(* PLC project plan_voie_railml, OpenIXl generator OpenIXL generator v0.1 *)
(* stored: companyURL https://github.com/Bleebop/IXL_project, creationDateTime 2026-09-27T16:06:12, modificationDateTime 2026-09-27T16:06:12 *)

TYPE TC : (NIL := -1, CDV10 := 1, CDV8 := 2, CDV6 := 3, CDV7 := 4, CDV9 := 5, CDV11 := 6, CDV13 := 7, CDV14 := 8, CDV12 := 9);
END_TYPE

TYPE SWITCH : (NIL := -1, SW2 := 1, SW1 := 2);
END_TYPE

TYPE SIGNAL : (NIL := -1, MRK13 := 1, MRK14 := 2, MRK15 := 3, MRK16 := 4);
END_TYPE

TYPE TRAIN_STATE : STRUCT
  exists : BOOL;
  rear_pos : TC;
  front_pos : TC;
  orientation : DIR;
  stopped : BOOL;
END_STRUCT;
END_TYPE

TYPE DIR : (NIL := -1, DOWN := 0, UP := 1);
END_TYPE

TYPE SW_POS_t : (NIL := -1, LEFT := 1, RIGHT := 2, INTERMEDIATE := 3);
END_TYPE

TYPE ENTRY_POINT_t : STRUCT
  tc : TC;
  orientation : DIR;
END_STRUCT;
END_TYPE

TYPE EXIT_POINT_t : STRUCT
  tc : TC;
  orientation : DIR;
END_STRUCT;
END_TYPE

TYPE ROUTE : (NIL := -1, ROUTE1 := 1, ROUTE2 := 2, ROUTE3 := 3);
END_TYPE

PROGRAM safety_PLC
  VAR
    route_state : ARRAY[1..const_g.nRoute] OF route_state;
    Approaching_train : ARRAY[1..const_g.nRoute] OF Approaching_train;
    switch_locked : ARRAY[1..const_g.nSwitch] OF BOOL;
    switch_required_left : ARRAY[1..const_g.nSwitch] OF BOOL;
    switch_required_right : ARRAY[1..const_g.nSwitch] OF BOOL;
  END_VAR
  VAR CONSTANT
    DELAY_DESTRUCT : ARRAY[1..const_g.nRoute] OF TIME := [TIME#99999s0ms, TIME#99999s0ms, TIME#99999s0ms];
  END_VAR
  VAR_OUTPUT
    route_open : ARRAY[1..const_g.nRoute] OF BOOL;
    route_entry_authorization : ARRAY[1..const_g.nRoute] OF BOOL;  (* The starting signal of the route can be opened to go through this route *)
    signal_open_maneuver : ARRAY[1..const_g.nSignal] OF BOOL;  (* Signal is opened for CBTC trains (downstream block occupation is ignored) *)
    switch_command_left : ARRAY[1..const_g.nSwitch] OF BOOL;
    switch_command_right : ARRAY[1..const_g.nSwitch] OF BOOL;
  END_VAR

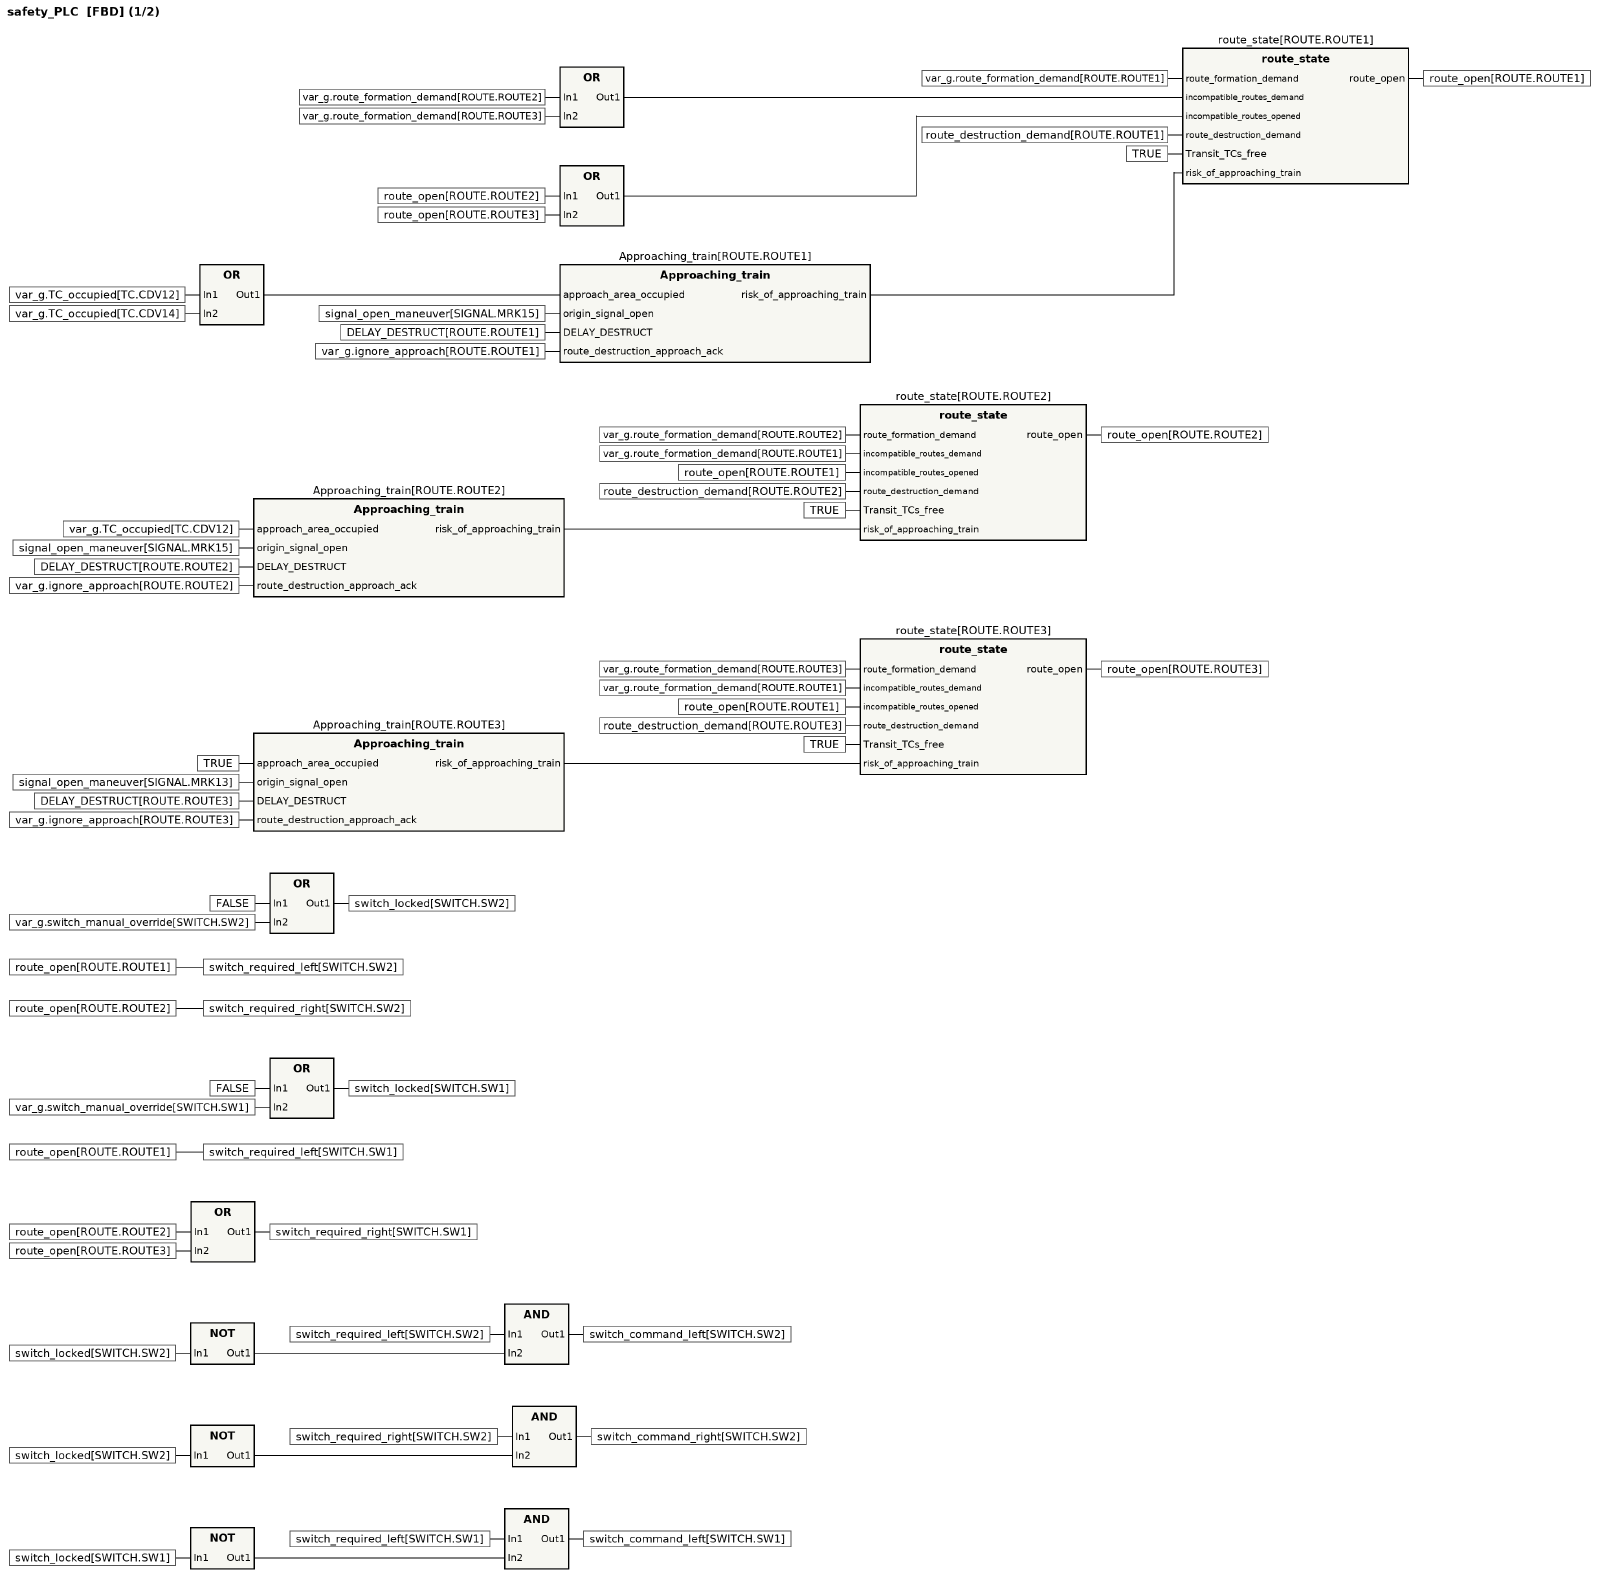
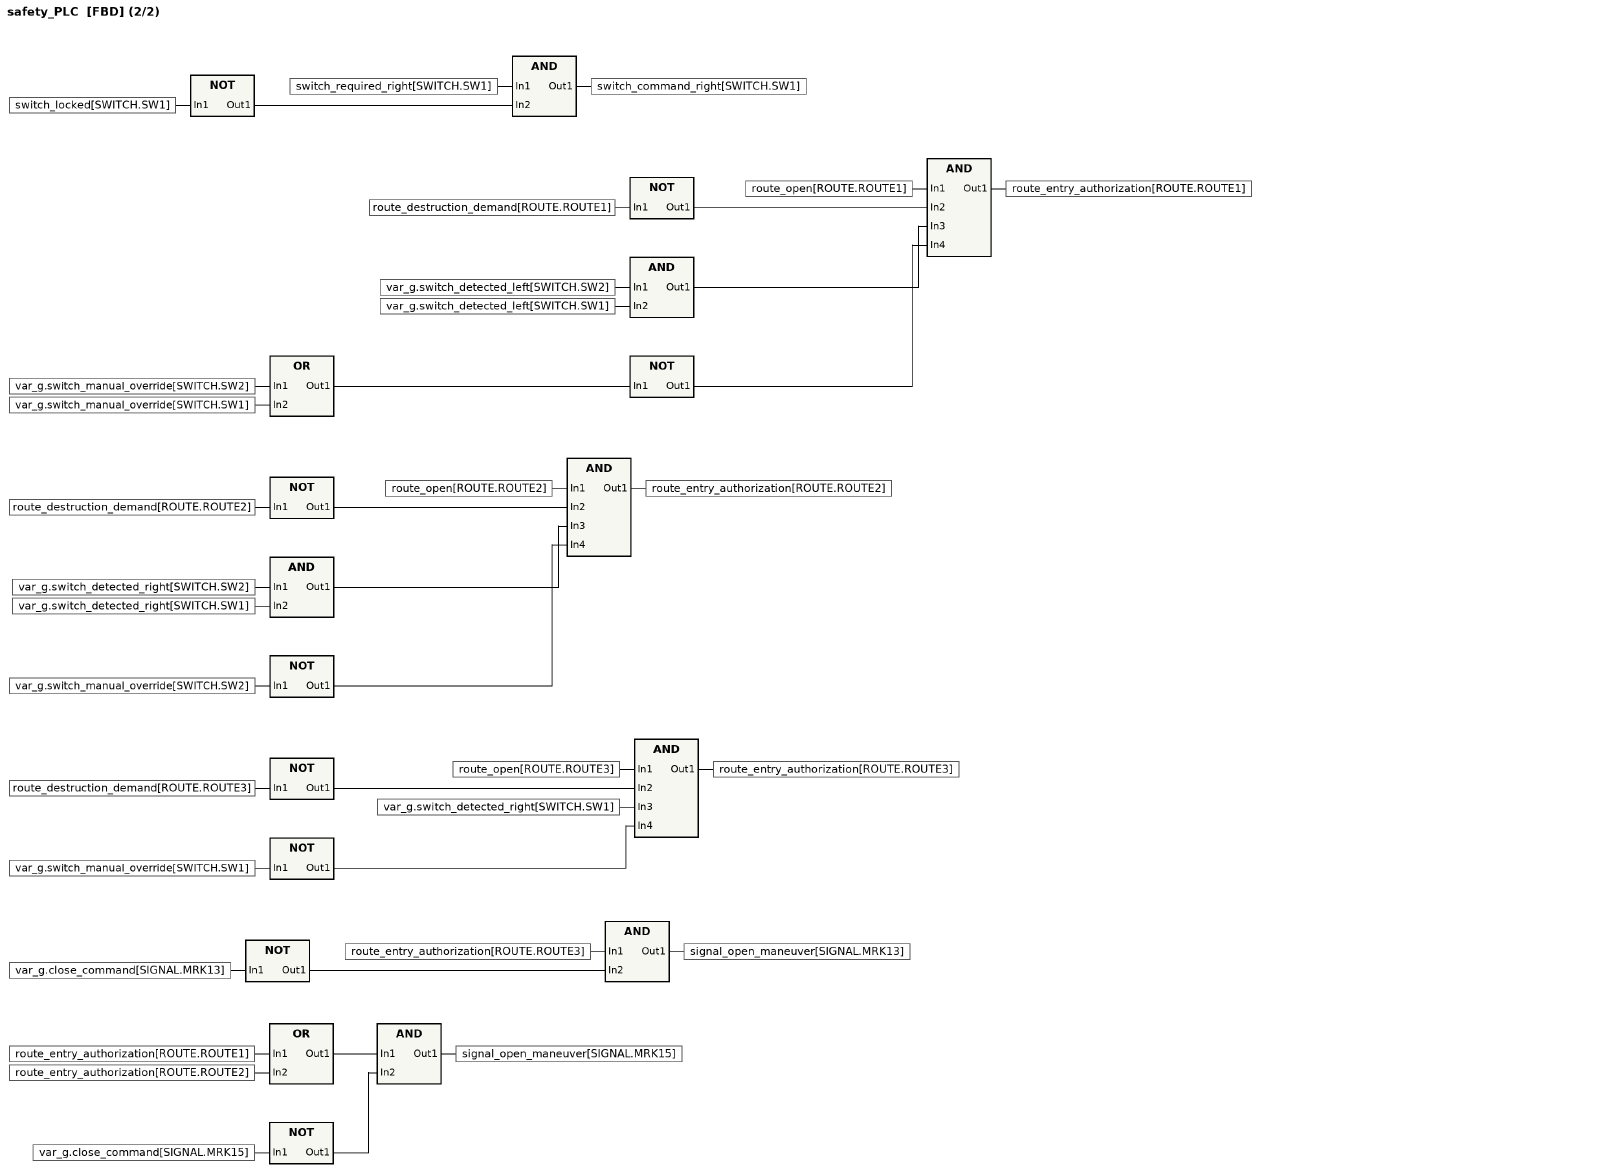
(* FBD diagram, written out as Structured Text *)
Approaching_train[ROUTE.ROUTE1](approach_area_occupied := var_g.TC_occupied[TC.CDV12] OR var_g.TC_occupied[TC.CDV14], origin_signal_open := signal_open_maneuver[SIGNAL.MRK15], DELAY_DESTRUCT := DELAY_DESTRUCT[ROUTE.ROUTE1], route_destruction_approach_ack := var_g.ignore_approach[ROUTE.ROUTE1]);
route_state[ROUTE.ROUTE1](route_formation_demand := var_g.route_formation_demand[ROUTE.ROUTE1], incompatible_routes_demand := var_g.route_formation_demand[ROUTE.ROUTE2] OR var_g.route_formation_demand[ROUTE.ROUTE3], incompatible_routes_opened := route_open[ROUTE.ROUTE2] OR route_open[ROUTE.ROUTE3], route_destruction_demand := route_destruction_demand[ROUTE.ROUTE1], Transit_TCs_free := TRUE, risk_of_approaching_train := Approaching_train[ROUTE.ROUTE1].risk_of_approaching_train);
route_open[ROUTE.ROUTE1] := route_state[ROUTE.ROUTE1].route_open;
Approaching_train[ROUTE.ROUTE2](approach_area_occupied := var_g.TC_occupied[TC.CDV12], origin_signal_open := signal_open_maneuver[SIGNAL.MRK15], DELAY_DESTRUCT := DELAY_DESTRUCT[ROUTE.ROUTE2], route_destruction_approach_ack := var_g.ignore_approach[ROUTE.ROUTE2]);
route_state[ROUTE.ROUTE2](route_formation_demand := var_g.route_formation_demand[ROUTE.ROUTE2], incompatible_routes_demand := var_g.route_formation_demand[ROUTE.ROUTE1], incompatible_routes_opened := route_open[ROUTE.ROUTE1], route_destruction_demand := route_destruction_demand[ROUTE.ROUTE2], Transit_TCs_free := TRUE, risk_of_approaching_train := Approaching_train[ROUTE.ROUTE2].risk_of_approaching_train);
route_open[ROUTE.ROUTE2] := route_state[ROUTE.ROUTE2].route_open;
Approaching_train[ROUTE.ROUTE3](approach_area_occupied := TRUE, origin_signal_open := signal_open_maneuver[SIGNAL.MRK13], DELAY_DESTRUCT := DELAY_DESTRUCT[ROUTE.ROUTE3], route_destruction_approach_ack := var_g.ignore_approach[ROUTE.ROUTE3]);
route_state[ROUTE.ROUTE3](route_formation_demand := var_g.route_formation_demand[ROUTE.ROUTE3], incompatible_routes_demand := var_g.route_formation_demand[ROUTE.ROUTE1], incompatible_routes_opened := route_open[ROUTE.ROUTE1], route_destruction_demand := route_destruction_demand[ROUTE.ROUTE3], Transit_TCs_free := TRUE, risk_of_approaching_train := Approaching_train[ROUTE.ROUTE3].risk_of_approaching_train);
route_open[ROUTE.ROUTE3] := route_state[ROUTE.ROUTE3].route_open;
switch_locked[SWITCH.SW2] := FALSE OR var_g.switch_manual_override[SWITCH.SW2];
switch_required_left[SWITCH.SW2] := route_open[ROUTE.ROUTE1];
switch_required_right[SWITCH.SW2] := route_open[ROUTE.ROUTE2];
switch_locked[SWITCH.SW1] := FALSE OR var_g.switch_manual_override[SWITCH.SW1];
switch_required_left[SWITCH.SW1] := route_open[ROUTE.ROUTE1];
switch_required_right[SWITCH.SW1] := route_open[ROUTE.ROUTE2] OR route_open[ROUTE.ROUTE3];
switch_command_left[SWITCH.SW2] := switch_required_left[SWITCH.SW2] AND NOT switch_locked[SWITCH.SW2];
switch_command_right[SWITCH.SW2] := switch_required_right[SWITCH.SW2] AND NOT switch_locked[SWITCH.SW2];
switch_command_left[SWITCH.SW1] := switch_required_left[SWITCH.SW1] AND NOT switch_locked[SWITCH.SW1];
switch_command_right[SWITCH.SW1] := switch_required_right[SWITCH.SW1] AND NOT switch_locked[SWITCH.SW1];
route_entry_authorization[ROUTE.ROUTE1] := route_open[ROUTE.ROUTE1] AND NOT route_destruction_demand[ROUTE.ROUTE1] AND var_g.switch_detected_left[SWITCH.SW2] AND var_g.switch_detected_left[SWITCH.SW1] AND NOT (var_g.switch_manual_override[SWITCH.SW2] OR var_g.switch_manual_override[SWITCH.SW1]);
route_entry_authorization[ROUTE.ROUTE2] := route_open[ROUTE.ROUTE2] AND NOT route_destruction_demand[ROUTE.ROUTE2] AND var_g.switch_detected_right[SWITCH.SW2] AND var_g.switch_detected_right[SWITCH.SW1] AND NOT var_g.switch_manual_override[SWITCH.SW2];
route_entry_authorization[ROUTE.ROUTE3] := route_open[ROUTE.ROUTE3] AND NOT route_destruction_demand[ROUTE.ROUTE3] AND var_g.switch_detected_right[SWITCH.SW1] AND NOT var_g.switch_manual_override[SWITCH.SW1];
signal_open_maneuver[SIGNAL.MRK13] := route_entry_authorization[ROUTE.ROUTE3] AND NOT var_g.close_command[SIGNAL.MRK13];
signal_open_maneuver[SIGNAL.MRK15] := (route_entry_authorization[ROUTE.ROUTE1] OR route_entry_authorization[ROUTE.ROUTE2]) AND NOT var_g.close_command[SIGNAL.MRK15];
END_PROGRAM

FUNCTION_BLOCK route_state
  VAR_INPUT
    route_formation_demand : BOOL;
    incompatible_routes_demand : BOOL;
    incompatible_routes_opened : BOOL;
    route_destruction_demand : BOOL;
    Transit_TCs_free : BOOL;
    risk_of_approaching_train : BOOL;
  END_VAR
  VAR
    SR_route : SR;
  END_VAR
  VAR_OUTPUT
    route_open : BOOL;
  END_VAR

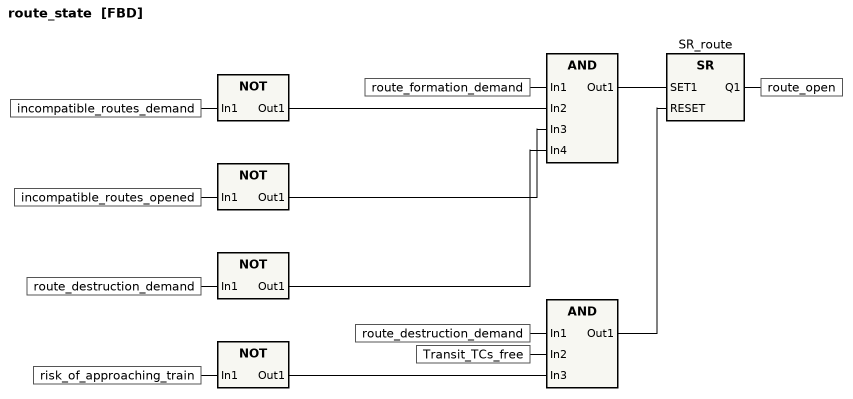
(* FBD diagram, written out as Structured Text *)
SR_route(SET1 := route_formation_demand AND NOT incompatible_routes_demand AND NOT incompatible_routes_opened AND NOT route_destruction_demand, RESET := route_destruction_demand AND Transit_TCs_free AND NOT risk_of_approaching_train);
route_open := SR_route.Q1;
END_FUNCTION_BLOCK

FUNCTION_BLOCK Approaching_train
  VAR_INPUT
    approach_area_occupied : BOOL;
    origin_signal_open : BOOL;
    DELAY_DESTRUCT : TIME;
    route_destruction_approach_ack : BOOL;
  END_VAR
  VAR_OUTPUT
    risk_of_approaching_train : BOOL;
  END_VAR
  VAR
    TON_approach_timer : TON;
    SR_approaching_train : SR;
  END_VAR

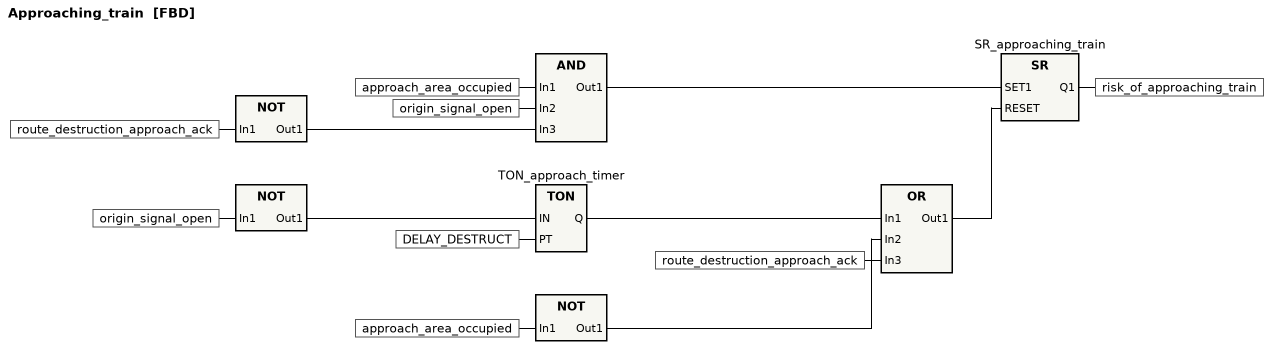
(* FBD diagram, written out as Structured Text *)
TON_approach_timer(IN := NOT origin_signal_open, PT := DELAY_DESTRUCT);
SR_approaching_train(SET1 := approach_area_occupied AND origin_signal_open AND NOT route_destruction_approach_ack, RESET := TON_approach_timer.Q OR NOT approach_area_occupied OR route_destruction_approach_ack);
risk_of_approaching_train := SR_approaching_train.Q1;
END_FUNCTION_BLOCK

CONFIGURATION Device
  RESOURCE Application ON PLC
    VAR_GLOBAL  (* var_g *)
      TC_occupied : ARRAY[1..const_g.nTC] OF BOOL;  (* /!\ safety critical /!\ *)
      switch_detected_left : ARRAY[1..const_g.nSwitch] OF BOOL;  (* /!\ safety critical /!\ *)
      switch_detected_right : ARRAY[1..const_g.nSwitch] OF BOOL;  (* /!\ safety critical /!\ *)
      switch_manual_override : ARRAY[1..const_g.nSwitch] OF BOOL;  (* Allows a switch to be moved on site /!\ safety critical /!\ *)
      close_command : ARRAY[1..const_g.nSignal] OF BOOL;  (* Force a signal to be closed *)
      ignore_TC_occupation : ARRAY[1..const_g.nTC] OF BOOL;  (* Allow to destruct a route even if this TC is occupied. /!\ safety critical /!\ *)
      ignore_approach : ARRAY[1..const_g.nRoute] OF BOOL;  (* Allow to destruct a route even if there is a risk of a train entering. /!\ safety critical /!\ *)
      route_formation_demand : ARRAY[1..const_g.nRoute] OF BOOL;
      route_destruction_demand : ARRAY[1..const_g.nRoute] OF BOOL;
    END_VAR
    VAR_GLOBAL CONSTANT  (* const_g *)
      nTC : INT := 9;  (* Track Circuits used by the IXL *)
      nRoute : INT := 3;  (* Routes that can be formed and destroyed *)
      nSwitch : INT := 2;
      nSignal : INT := 4;
    END_VAR
    TASK MainTask(INTERVAL := T#50ms, PRIORITY := 1);
    PROGRAM safety_PLC WITH MainTask : safety_PLC;
  END_RESOURCE
END_CONFIGURATION
